(* CODESYS project MateusBastos_TalitaFelix (1).project

Project tree, tasks and I/O mapping:
  Device : CODESYS Control Win V3, 3S - Smart Software Solutions GmbH, order no. 305021, version 3.5.11.40
    application Application
      libraries: Standard, * (System)
      task MainTask (cyclic, interval t#10ms, priority 1) calls Main, Doca2_automatico, Doca1_manual, Doca2_manual, Doca1_automatico
      task Simulacao (cyclic, interval t#20ms, priority 1) calls Simulacao_Valores, Doca2_Simulacao, Gasolina_Simulacao, Doca1_Simulacao
      program Doca1_manual [SFC]
      global variables GVL
      program Doca2_manual [SFC]
      program Doca1_automatico [SFC]
      program Doca2_automatico [SFC]
      program Main [ST]
      Simulacao/
        program Doca2_Simulacao [ST]
        program Simulacao_Valores [ST]
        program Doca1_Simulacao [ST]
        program Gasolina_Simulacao [ST]
      program Emergencia [ST]
*)

// Device/Application/GVL
{attribute 'qualified_only'}
VAR_GLOBAL
// Sensores Analógicos - Entradas
LT_S01 : REAL;   // Sensor de porcentagem de etanol no silo 1
LT_S02 : REAL;   // Sensor de porcentagem de gasolina no silo 2
LT_S03 : REAL;   // Sensor de porcentagem de etanol no silo 3

// Sensores Discretos - Entradas
LSH_S01 : BOOL;  // Sensor de quantidade alta de combustível no silo 1
LSL_S01 : BOOL;  // Sensor de quantidade baixa de combustível no silo 1
LSH_S02 : BOOL;  // Sensor de quantidade alta de combustível no silo 2
LSL_S02 : BOOL;  // Sensor de quantidade baixa de combustível no silo 2
LSH_S03 : BOOL;  // Sensor de quantidade alta de combustível no silo 3
LSL_S03 : BOOL;  // Sensor de quantidade baixa de combustível no silo 3

// Atuadores Discretos - Saídas
VA_S01 : BOOL;   // Válvula de admissão de etanol no silo 1
VA_S02 : BOOL;   // Válvula de admissão de gasolina no silo 2
VA_S03 : BOOL;   // Válvula de admissão de etanol no silo 3
VS_S01 : BOOL;   // Válvula de admissão de etanol no tanque
VS_S02_1 : BOOL; // Válvula de admissão de gasolina no tanque (primeira seção)
VS_S02_2 : BOOL; // Válvula de admissão de gasolina no tanque (segunda seção)
VS_S03 : BOOL;   // Válvula de admissão de etanol no tanque
VC_TQ2 : BOOL;   // Válvula de saída do combustível para a mangueira (tanque 2)
VC_TQ1 : BOOL;   // Válvula de saída do combustível para a mangueira (tanque 1)
M1 : BOOL;       // Misturador 1
M2 : BOOL;       // Misturador 2
B_R1 : BOOL;     // Bomba de Etanol
B_R2 : BOOL;     // Bomba de Gasolina
C_D1 : BOOL;     // Cancela 1
C_D2 : BOOL;     // Cancela 2

// Interface - máquina
liga_manual: BOOL;
liga_auto: BOOL;
desliga: BOOL;
emergencia: BOOL;
rearme: BOOL;
Y_C_D1: BOOL;
Y_M_D1: BOOL;
Y_C_D2: BOOL;
Y_M_D2: BOOL;
etanol_D1: BOOL;
gasolina_p_D1: BOOL;
gasolina_n_D1: BOOL;
etanol_D2: BOOL;
gasolina_p_D2: BOOL;
gasolina_n_D2: BOOL;
//etanol_cheio: BOOL;
//gasolina_cheio: BOOL;
//timer_misturador: BOOL;
caminhao1_cheio: BOOL;
caminhao2_cheio: BOOL;
alarme_D1: BOOL;
alarme_D2: BOOL;

V_R_Etanol : INT := 200; //Vazao Reservatorio Etanol
V_R_Gasolina : INT := 200; //Vazao Reservatorio Gasolina
V_S01_TQ1 : INT := 100; // Vazão do Silo para o Tanque
V_S02_TQ : INT := 100; // Vazão DO Silo para o Tanque
V_S03_TQ2 : INT := 100; // Vazão DO Silo para o Tanque
TQ1_C : INT := 100;
TQ2_C : INT := 100;

volume_S01 : REAL := 50000;
volume_S02 : REAL := 50000;
volume_S03 : REAL := 50000;

volume_C1 : REAL := 0;
volume_C2 : REAL := 0;

volume_TQ1 : REAL := 0;
volume_TQ2 : REAL := 0;

volume_gasolina_C1 : REAL := 0;
volume_gasolina_C2 : REAL := 0;

volume_etanol_C1 : REAL := 0;
volume_etanol_C2 : REAL := 0;

PREMIUM : BOOL; // SE PREMIUM, GASOLINA PREMIUM.
ETANOL : BOOL; //EXCLUIR ESSA VARIAVEL

modo_op : BOOL; //Modo de operação atual do programa
switch : BOOl; //Modo de operação que o operador definiu

END_VAR

// Device/Application/Main
PROGRAM Main


// Desliga foi ativado
IF GVL.desliga THEN
	// Para a operação de todas as docas
	Doca1_manual.Ligar := FALSE;
	Doca2_manual.Ligar := FALSE;
	Doca1_automatico.Ligar := FALSE;
	Doca2_automatico.Ligar := FALSE;

// Emergência foi ativada
ELSIF GVL.emergencia AND NOT GVL.Rearme AND NOT GVL.modo_op THEN
	// Para a operação de todas as docas
	Emergencia.Ligar := TRUE;
	Doca1_manual.Ligar := FALSE;
	Doca2_manual.Ligar := FALSE;

ELSIF GVL.rearme AND NOT GVL.modo_op THEN
	Emergencia.Ligar := FALSE;
	Doca1_manual.Ligar := TRUE;
	Doca2_manual.Ligar := TRUE;

ELSIF GVL.emergencia AND NOT GVL.Rearme AND GVL.modo_op THEN
	// Para a operação de todas as docas
	Emergencia.Ligar := TRUE;
	Doca1_automatico.Ligar := FALSE;
	Doca2_automatico.Ligar := FALSE;

ELSIF GVL.rearme AND GVL.modo_op THEN
	Emergencia.Ligar := FALSE;
	Doca1_automatico.Ligar := TRUE;
	Doca2_automatico.Ligar := TRUE;

// Seleção do modo de operação e liga	
ELSE
	// Se o modo de operação for manual e o operador requisitar o modo automático, o modo_op será trocado se não houver caminhões na doca e todas as válvulas estiverem fechadas
	IF GVL.modo_op = 0 AND GVL.switch = 1 THEN
		IF (Doca1_manual.Init.x AND Doca2_manual.Init.x) OR (NOT Doca1_manual.Ligar AND NOT Doca2_manual.Ligar) OR Emergencia.Ligar THEN
			GVL.modo_op := 1;
		END_IF	
	END_IF
	
	// Se o modo de operação for automático e o operador requisitar o modo manual, o modo_op será trocado se o processo estiver desligago ou em estado de emergência
	IF GVL.modo_op = 1 AND GVL.switch = 0 THEN
		IF NOT GVL.liga_auto OR Emergencia.Ligar THEN
			GVL.modo_op := 0;
		END_IF	
	END_IF
	
	IF GVL.liga_manual AND NOT GVL.modo_op THEN
		// Inicia a operação manual das duas docas
		Doca1_manual.Ligar := TRUE;
		Doca2_manual.Ligar := TRUE;
		Doca1_automatico.Ligar := FALSE;
		Doca2_automatico.Ligar := FALSE;
		
	ELSIF GVL.liga_auto AND GVL.modo_op THEN
		// Inicia a operação automática das duas docas
		Doca1_manual.Ligar := FALSE;
		Doca2_manual.Ligar := FALSE;
		Doca1_automatico.Ligar := TRUE;
		Doca2_automatico.Ligar := TRUE;
		
	END_IF
END_IF

END_PROGRAM

// Device/Application/Doca1_manual
PROGRAM Doca1_manual
VAR_INPUT
	Ligar : BOOL;
END_VAR

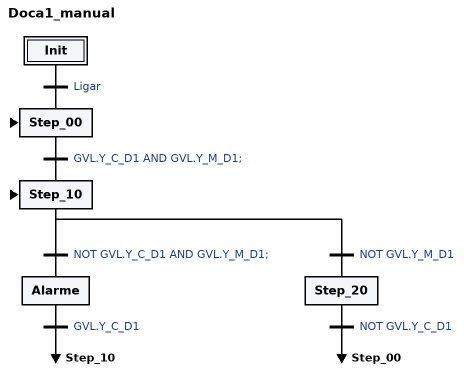
INITIAL_STEP Init:
END_STEP
TRANSITION FROM Init TO Step_00
    := Ligar;
END_TRANSITION
STEP Step_00:
END_STEP
TRANSITION FROM Step_00 TO Step_10
    := GVL.Y_C_D1 AND GVL.Y_M_D1;
END_TRANSITION
STEP Step_10:
END_STEP
TRANSITION FROM Step_10 TO Alarme
    := NOT GVL.Y_C_D1 AND GVL.Y_M_D1;
END_TRANSITION
STEP Alarme:
END_STEP
TRANSITION FROM Alarme TO Step_10
    := GVL.Y_C_D1;
END_TRANSITION
TRANSITION FROM Step_10 TO Step_20
    := NOT GVL.Y_M_D1;
END_TRANSITION
STEP Step_20:
END_STEP
TRANSITION FROM Step_20 TO Step_00
    := NOT GVL.Y_C_D1;
END_TRANSITION

END_PROGRAM

// Device/Application/Doca2_manual
PROGRAM Doca2_manual
VAR_INPUT
	Ligar : BOOL;
END_VAR

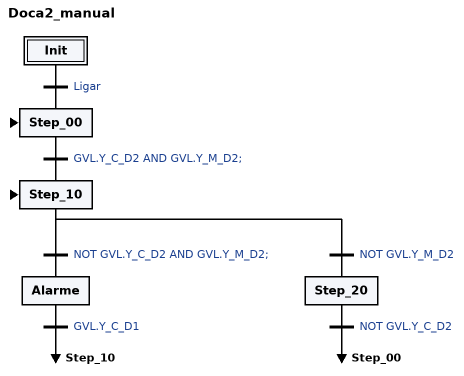
INITIAL_STEP Init:
END_STEP
TRANSITION FROM Init TO Step_00
    := Ligar;
END_TRANSITION
STEP Step_00:
END_STEP
TRANSITION FROM Step_00 TO Step_10
    := GVL.Y_C_D2 AND GVL.Y_M_D2;
END_TRANSITION
STEP Step_10:
END_STEP
TRANSITION FROM Step_10 TO Alarme
    := NOT GVL.Y_C_D2 AND GVL.Y_M_D2;
END_TRANSITION
STEP Alarme:
END_STEP
TRANSITION FROM Alarme TO Step_10
    := GVL.Y_C_D1;
END_TRANSITION
TRANSITION FROM Step_10 TO Step_20
    := NOT GVL.Y_M_D2;
END_TRANSITION
STEP Step_20:
END_STEP
TRANSITION FROM Step_20 TO Step_00
    := NOT GVL.Y_C_D2;
END_TRANSITION

END_PROGRAM

// Device/Application/Doca1_automatico
	PROGRAM Doca1_automatico

VAR_INPUT
	Ligar : BOOL;
	etanol_cheio: BOOL;
	gasolina_cheio: BOOL;
END_VAR

VAR
	
END_VAR

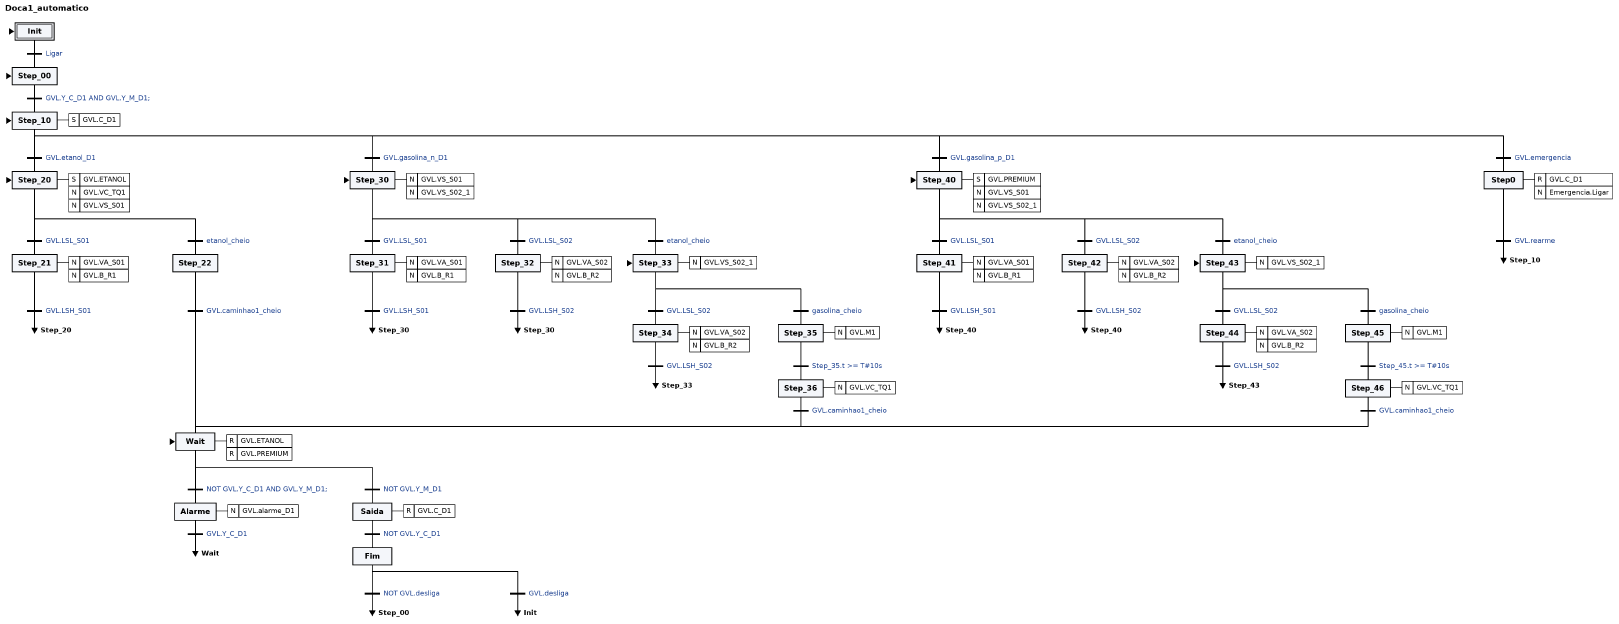
INITIAL_STEP Init:
END_STEP
TRANSITION FROM Init TO Step_00
    := Ligar;
END_TRANSITION
STEP Step_00:
END_STEP
TRANSITION FROM Step_00 TO Step_10
    := GVL.Y_C_D1 AND GVL.Y_M_D1;
END_TRANSITION
STEP Step_10:
    GVL.C_D1(S);
END_STEP
TRANSITION FROM Step_10 TO Step_20
    := GVL.etanol_D1;
END_TRANSITION
STEP Step_20:
    GVL.ETANOL(S);
    GVL.VC_TQ1(N);
    GVL.VS_S01(N);
END_STEP
TRANSITION FROM Step_20 TO Step_21
    := GVL.LSL_S01;
END_TRANSITION
STEP Step_21:
    GVL.VA_S01(N);
    GVL.B_R1(N);
END_STEP
TRANSITION FROM Step_21 TO Step_20
    := GVL.LSH_S01;
END_TRANSITION
TRANSITION FROM Step_20 TO Step_22
    := etanol_cheio;
END_TRANSITION
STEP Step_22:
END_STEP
TRANSITION FROM Step_22 TO Wait
    := GVL.caminhao1_cheio;
END_TRANSITION
TRANSITION FROM Step_10 TO Step_30
    := GVL.gasolina_n_D1;
END_TRANSITION
STEP Step_30:
    GVL.VS_S01(N);
    GVL.VS_S02_1(N);
END_STEP
TRANSITION FROM Step_30 TO Step_31
    := GVL.LSL_S01;
END_TRANSITION
STEP Step_31:
    GVL.VA_S01(N);
    GVL.B_R1(N);
END_STEP
TRANSITION FROM Step_31 TO Step_30
    := GVL.LSH_S01;
END_TRANSITION
TRANSITION FROM Step_30 TO Step_32
    := GVL.LSL_S02;
END_TRANSITION
STEP Step_32:
    GVL.VA_S02(N);
    GVL.B_R2(N);
END_STEP
TRANSITION FROM Step_32 TO Step_30
    := GVL.LSH_S02;
END_TRANSITION
TRANSITION FROM Step_30 TO Step_33
    := etanol_cheio;
END_TRANSITION
STEP Step_33:
    GVL.VS_S02_1(N);
END_STEP
TRANSITION FROM Step_33 TO Step_34
    := GVL.LSL_S02;
END_TRANSITION
STEP Step_34:
    GVL.VA_S02(N);
    GVL.B_R2(N);
END_STEP
TRANSITION FROM Step_34 TO Step_33
    := GVL.LSH_S02;
END_TRANSITION
TRANSITION FROM Step_33 TO Step_35
    := gasolina_cheio;
END_TRANSITION
STEP Step_35:
    GVL.M1(N);
END_STEP
TRANSITION FROM Step_35 TO Step_36
    := Step_35.t >= T#10s;
END_TRANSITION
STEP Step_36:
    GVL.VC_TQ1(N);
END_STEP
TRANSITION FROM Step_36 TO Wait
    := GVL.caminhao1_cheio;
END_TRANSITION
TRANSITION FROM Step_10 TO Step_40
    := GVL.gasolina_p_D1;
END_TRANSITION
STEP Step_40:
    GVL.PREMIUM(S);
    GVL.VS_S01(N);
    GVL.VS_S02_1(N);
END_STEP
TRANSITION FROM Step_40 TO Step_41
    := GVL.LSL_S01;
END_TRANSITION
STEP Step_41:
    GVL.VA_S01(N);
    GVL.B_R1(N);
END_STEP
TRANSITION FROM Step_41 TO Step_40
    := GVL.LSH_S01;
END_TRANSITION
TRANSITION FROM Step_40 TO Step_42
    := GVL.LSL_S02;
END_TRANSITION
STEP Step_42:
    GVL.VA_S02(N);
    GVL.B_R2(N);
END_STEP
TRANSITION FROM Step_42 TO Step_40
    := GVL.LSH_S02;
END_TRANSITION
TRANSITION FROM Step_40 TO Step_43
    := etanol_cheio;
END_TRANSITION
STEP Step_43:
    GVL.VS_S02_1(N);
END_STEP
TRANSITION FROM Step_43 TO Step_44
    := GVL.LSL_S02;
END_TRANSITION
STEP Step_44:
    GVL.VA_S02(N);
    GVL.B_R2(N);
END_STEP
TRANSITION FROM Step_44 TO Step_43
    := GVL.LSH_S02;
END_TRANSITION
TRANSITION FROM Step_43 TO Step_45
    := gasolina_cheio;
END_TRANSITION
STEP Step_45:
    GVL.M1(N);
END_STEP
TRANSITION FROM Step_45 TO Step_46
    := Step_45.t >= T#10s;
END_TRANSITION
STEP Step_46:
    GVL.VC_TQ1(N);
END_STEP
TRANSITION FROM Step_46 TO Wait
    := GVL.caminhao1_cheio;
END_TRANSITION
TRANSITION FROM Step_10 TO Step0
    := GVL.emergencia;
END_TRANSITION
STEP Step0:
    GVL.C_D1(R);
    Emergencia.Ligar(N);
END_STEP
TRANSITION FROM Step0 TO Step_10
    := GVL.rearme;
END_TRANSITION
STEP Wait:
    GVL.ETANOL(R);
    GVL.PREMIUM(R);
END_STEP
TRANSITION FROM Wait TO Alarme
    := NOT GVL.Y_C_D1 AND GVL.Y_M_D1;
END_TRANSITION
STEP Alarme:
    GVL.alarme_D1(N);
END_STEP
TRANSITION FROM Alarme TO Wait
    := GVL.Y_C_D1;
END_TRANSITION
TRANSITION FROM Wait TO Saida
    := NOT GVL.Y_M_D1;
END_TRANSITION
STEP Saida:
    GVL.C_D1(R);
END_STEP
TRANSITION FROM Saida TO Fim
    := NOT GVL.Y_C_D1;
END_TRANSITION
STEP Fim:
END_STEP
TRANSITION FROM Fim TO Step_00
    := NOT GVL.desliga;
END_TRANSITION
TRANSITION FROM Fim TO Init
    := GVL.desliga;
END_TRANSITION

END_PROGRAM

// Device/Application/Doca2_automatico
PROGRAM Doca2_automatico
VAR_INPUT
	Ligar : BOOL;
	etanol_cheio: BOOL;
	gasolina_cheio: BOOL;
END_VAR

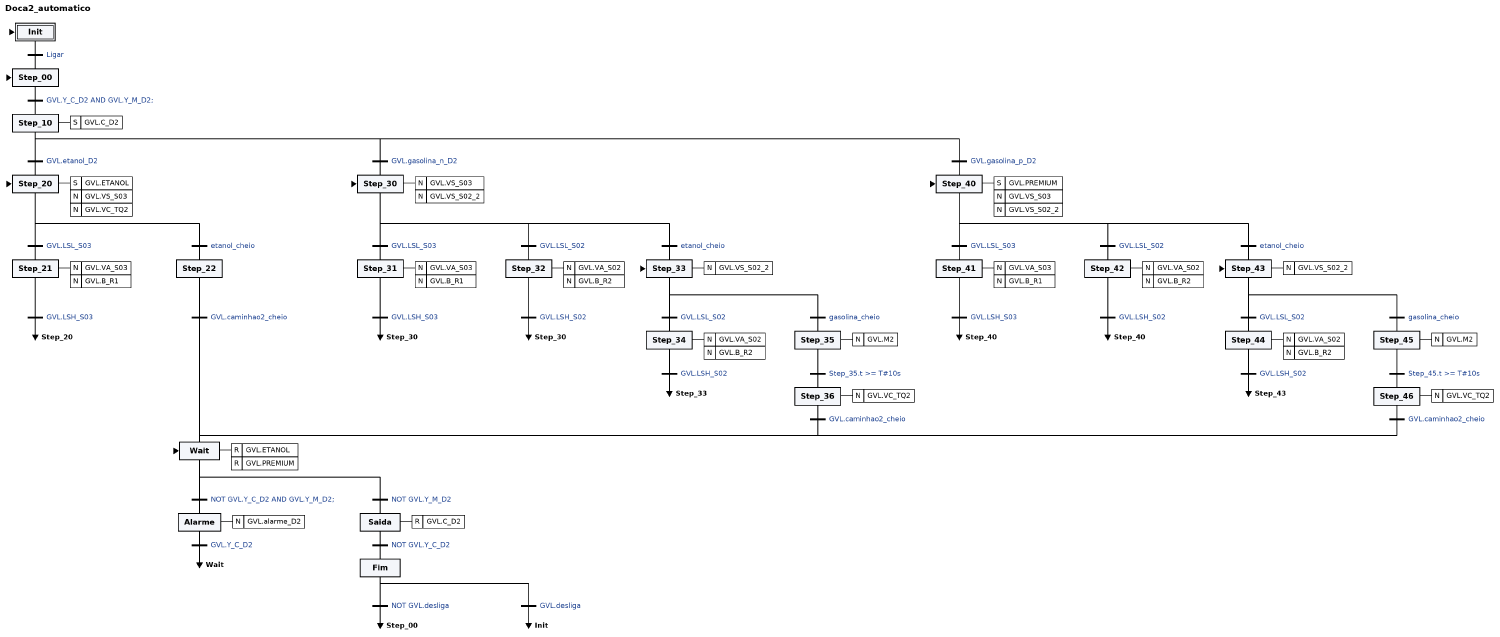
INITIAL_STEP Init:
END_STEP
TRANSITION FROM Init TO Step_00
    := Ligar;
END_TRANSITION
STEP Step_00:
END_STEP
TRANSITION FROM Step_00 TO Step_10
    := GVL.Y_C_D2 AND GVL.Y_M_D2;
END_TRANSITION
STEP Step_10:
    GVL.C_D2(S);
END_STEP
TRANSITION FROM Step_10 TO Step_20
    := GVL.etanol_D2;
END_TRANSITION
STEP Step_20:
    GVL.ETANOL(S);
    GVL.VS_S03(N);
    GVL.VC_TQ2(N);
END_STEP
TRANSITION FROM Step_20 TO Step_21
    := GVL.LSL_S03;
END_TRANSITION
STEP Step_21:
    GVL.VA_S03(N);
    GVL.B_R1(N);
END_STEP
TRANSITION FROM Step_21 TO Step_20
    := GVL.LSH_S03;
END_TRANSITION
TRANSITION FROM Step_20 TO Step_22
    := etanol_cheio;
END_TRANSITION
STEP Step_22:
END_STEP
TRANSITION FROM Step_22 TO Wait
    := GVL.caminhao2_cheio;
END_TRANSITION
TRANSITION FROM Step_10 TO Step_30
    := GVL.gasolina_n_D2;
END_TRANSITION
STEP Step_30:
    GVL.VS_S03(N);
    GVL.VS_S02_2(N);
END_STEP
TRANSITION FROM Step_30 TO Step_31
    := GVL.LSL_S03;
END_TRANSITION
STEP Step_31:
    GVL.VA_S03(N);
    GVL.B_R1(N);
END_STEP
TRANSITION FROM Step_31 TO Step_30
    := GVL.LSH_S03;
END_TRANSITION
TRANSITION FROM Step_30 TO Step_32
    := GVL.LSL_S02;
END_TRANSITION
STEP Step_32:
    GVL.VA_S02(N);
    GVL.B_R2(N);
END_STEP
TRANSITION FROM Step_32 TO Step_30
    := GVL.LSH_S02;
END_TRANSITION
TRANSITION FROM Step_30 TO Step_33
    := etanol_cheio;
END_TRANSITION
STEP Step_33:
    GVL.VS_S02_2(N);
END_STEP
TRANSITION FROM Step_33 TO Step_34
    := GVL.LSL_S02;
END_TRANSITION
STEP Step_34:
    GVL.VA_S02(N);
    GVL.B_R2(N);
END_STEP
TRANSITION FROM Step_34 TO Step_33
    := GVL.LSH_S02;
END_TRANSITION
TRANSITION FROM Step_33 TO Step_35
    := gasolina_cheio;
END_TRANSITION
STEP Step_35:
    GVL.M2(N);
END_STEP
TRANSITION FROM Step_35 TO Step_36
    := Step_35.t >= T#10s;
END_TRANSITION
STEP Step_36:
    GVL.VC_TQ2(N);
END_STEP
TRANSITION FROM Step_36 TO Wait
    := GVL.caminhao2_cheio;
END_TRANSITION
TRANSITION FROM Step_10 TO Step_40
    := GVL.gasolina_p_D2;
END_TRANSITION
STEP Step_40:
    GVL.PREMIUM(S);
    GVL.VS_S03(N);
    GVL.VS_S02_2(N);
END_STEP
TRANSITION FROM Step_40 TO Step_41
    := GVL.LSL_S03;
END_TRANSITION
STEP Step_41:
    GVL.VA_S03(N);
    GVL.B_R1(N);
END_STEP
TRANSITION FROM Step_41 TO Step_40
    := GVL.LSH_S03;
END_TRANSITION
TRANSITION FROM Step_40 TO Step_42
    := GVL.LSL_S02;
END_TRANSITION
STEP Step_42:
    GVL.VA_S02(N);
    GVL.B_R2(N);
END_STEP
TRANSITION FROM Step_42 TO Step_40
    := GVL.LSH_S02;
END_TRANSITION
TRANSITION FROM Step_40 TO Step_43
    := etanol_cheio;
END_TRANSITION
STEP Step_43:
    GVL.VS_S02_2(N);
END_STEP
TRANSITION FROM Step_43 TO Step_44
    := GVL.LSL_S02;
END_TRANSITION
STEP Step_44:
    GVL.VA_S02(N);
    GVL.B_R2(N);
END_STEP
TRANSITION FROM Step_44 TO Step_43
    := GVL.LSH_S02;
END_TRANSITION
TRANSITION FROM Step_43 TO Step_45
    := gasolina_cheio;
END_TRANSITION
STEP Step_45:
    GVL.M2(N);
END_STEP
TRANSITION FROM Step_45 TO Step_46
    := Step_45.t >= T#10s;
END_TRANSITION
STEP Step_46:
    GVL.VC_TQ2(N);
END_STEP
TRANSITION FROM Step_46 TO Wait
    := GVL.caminhao2_cheio;
END_TRANSITION
STEP Wait:
    GVL.ETANOL(R);
    GVL.PREMIUM(R);
END_STEP
TRANSITION FROM Wait TO Alarme
    := NOT GVL.Y_C_D2 AND GVL.Y_M_D2;
END_TRANSITION
STEP Alarme:
    GVL.alarme_D2(N);
END_STEP
TRANSITION FROM Alarme TO Wait
    := GVL.Y_C_D2;
END_TRANSITION
TRANSITION FROM Wait TO Saida
    := NOT GVL.Y_M_D2;
END_TRANSITION
STEP Saida:
    GVL.C_D2(R);
END_STEP
TRANSITION FROM Saida TO Fim
    := NOT GVL.Y_C_D2;
END_TRANSITION
STEP Fim:
END_STEP
TRANSITION FROM Fim TO Step_00
    := NOT GVL.desliga;
END_TRANSITION
TRANSITION FROM Fim TO Init
    := GVL.desliga;
END_TRANSITION

END_PROGRAM

// Device/Application/Emergencia
PROGRAM Emergencia

VAR_INPUT
	Ligar : BOOL;
END_VAR

IF Ligar THEN
	GVL.VA_S01 := FALSE;   
	GVL.VA_S02 := FALSE;
	GVL.VA_S03 := FALSE;
	GVL.VS_S01 := FALSE;
	GVL.VS_S02_1 := FALSE;
	GVL.VS_S02_2 := FALSE;
	GVL.VS_S03 := FALSE;
	GVL.VC_TQ2 := FALSE;
	GVL.VC_TQ1 := FALSE;
	GVL.M1 := FALSE;
	GVL.M2 := FALSE;
	GVL.B_R1 := FALSE;
	//GVL.B_R2 := FALSE;
END_IF

END_PROGRAM

// Device/Application/Simulacao/Simulacao_Valores
PROGRAM Simulacao_Valores
VAR
	Volume_gasolina_comum : REAL := 25000 * 0.75;
	Volume_etanol_comum : REAL := 25000 * 0.25;
	Volume_gasolina_premium : REAL := 25000 * 0.73;
	Volume_etanol_premium : REAL := 25000 * 0.27;
END_VAR

IF GVL.volume_C1 >= 25000 THEN//AND GVL.volume_gasolina_C1 = 0 THEN
	Doca1_automatico.etanol_cheio := TRUE;
	GVL.caminhao1_cheio := TRUE;
	
	GVL.volume_etanol_C1 := 0;
	GVL.volume_gasolina_C1 := 0;
	
ELSIF GVL.volume_S01 <= 5000 THEN
	GVL.LSL_S01 := TRUE;
	GVL.LSH_S01 := FALSE;
	
ELSIF  GVL.volume_S02 <= 5000 THEN
	GVL.LSL_S02 := TRUE;
	GVL.LSH_S02 := FALSE;

ELSIF GVL.volume_S02 >= 45000 THEN
	GVL.LSH_S02 := TRUE;
	GVL.LSL_S02 := FALSE;
	
ELSIF GVL.volume_S01 >= 45000 THEN
	GVL.LSH_S01 := TRUE;
	GVL.LSL_S01 := FALSE;

ELSIF GVL.volume_etanol_C1 >= Volume_etanol_premium AND NOT (GVL.volume_gasolina_C1 >= Volume_gasolina_premium) AND GVL.PREMIUM THEN // PODE GERAR UM FUTURO PROBLEMA
	Doca1_automatico.etanol_cheio := TRUE;
	
ELSIF GVL.volume_gasolina_C1 >= Volume_gasolina_premium AND NOT GVL.M1 AND GVL.PREMIUM THEN // PODE GERAR UM PROBLEMA NO FUTURO
	Doca1_automatico.gasolina_cheio := TRUE;	
	
ELSIF GVL.volume_etanol_C1 >= Volume_etanol_comum AND NOT (GVL.volume_gasolina_C1 >= Volume_gasolina_comum) AND NOT GVL.PREMIUM THEN // PODE GERAR UM FUTURO PROBLEMA
	Doca1_automatico.etanol_cheio := TRUE;
	
ELSIF GVL.volume_gasolina_C1 >= Volume_gasolina_comum AND NOT GVL.M1 AND NOT GVL.PREMIUM THEN // PODE GERAR UM PROBLEMA NO FUTURO
	Doca1_automatico.gasolina_cheio := TRUE;
	
ELSIF GVL.M1 THEN
	GVL.volume_etanol_C1 := 0;
	GVL.volume_gasolina_C1 := 0;
	
ELSE
	GVL.LSL_S01 := FALSE;
	GVL.caminhao1_cheio := FALSE;
	Doca1_automatico.gasolina_cheio := FALSE;
	Doca1_automatico.etanol_cheio := FALSE;
	GVL.LSH_S01 := FALSE;
END_IF

END_PROGRAM

// Device/Application/Simulacao/Doca2_Simulacao
PROGRAM Doca2_Simulacao
VAR
END_VAR

IF NOT GVL.emergencia THEN
	//Estado  20 & //Estado 31 & //Estado 41 & //Estado 34 & //Estado 44
	IF GVL.VA_S03 AND GVL.B_R1 AND GVL.C_D2 THEN
	// Enchendo o Silo 01 de Etanol - STEP_21
		GVL.volume_S03 := GVL.volume_S03 + GVL.V_R_Etanol;
	
		GVL.volume_TQ2 := GVL.volume_TQ2;
		
		GVL.volume_C2 := GVL.volume_C2;
		
	//Estado  20	
	ELSIF GVL.VA_S02 AND GVL.B_R2 AND (GVL.ETANOL OR NOT GVL.Y_C_D1) THEN // Caso em que o somente a doca 2 está utilizando gasolina
		GVL.volume_S02 := GVL.volume_S02 + GVL.V_R_Gasolina;
		
	ELSIF GVL.VS_S03 AND GVL.C_D2 AND NOT GVL.VS_S02_2 AND GVL.VC_TQ2 THEN
	// Enchendo o Tanque 1 & Esvaziando o Silo 01 - STEP_20
		GVL.volume_S03 := GVL.volume_S03 - GVL.V_S03_TQ2;
		
		GVL.volume_TQ2 := GVL.volume_TQ2 + GVL.TQ2_C - GVL.V_S03_TQ2;
		
		GVL.volume_C2 := GVL.volume_C2 + GVL.TQ2_C;
		
	//Estado 30	- STEP_30 e STEP_40
	ELSIF GVL.VS_S03 AND GVL.VS_S02_2 AND GVL.C_D2 THEN
	// Enchendo o TQ 1 && Esvaziando o Silo 01 && Esvaziando o Silo 02
	
	//Situação em que começo a encher o tanque de gasolina e de etanol simultaneamente
	
		GVL.volume_S03 := GVL.volume_S03 - GVL.V_S03_TQ2; // Diminuo o volume do Silo 3
		
		GVL.volume_S02 := GVL.volume_S02 - GVL.V_S02_TQ; // Diminuo o volume do Silo 2
		
		GVL.volume_C2 := GVL.volume_C2; // Mantenho o volume do caminhão constante
		
		GVL.volume_TQ2 := GVL.volume_TQ2 + GVL.V_S02_TQ + GVL.V_S03_TQ2; // Aumento o volume do tanque 1
		
		GVL.volume_gasolina_C2 := GVL.volume_gasolina_C2 + GVL.V_S02_TQ; // Aumento a contagem da gasolina que está entrando no tanque
		
		GVL.volume_etanol_C2 := GVL.volume_etanol_C2 + GVL.V_S03_TQ2; // Aumento a contagem de etanol que está entrando no tanque
		
	//Estado 33 & Estado 43 - STEP_33
	ELSIF GVL.VS_S02_2 AND NOT GVL.VC_TQ2 AND GVL.C_D2 THEN
		GVL.volume_S02 := GVL.volume_S02 - GVL.V_S02_TQ;	
		
		GVL.volume_C2 := GVL.volume_C2;
		
		GVL.volume_TQ2 := GVL.volume_TQ2 + GVL.V_S02_TQ;
		
		GVL.volume_gasolina_C2 := GVL.volume_gasolina_C2 + GVL.V_S02_TQ;
		
	//Estado 35 & //Estado 45
	ELSIF GVL.M2 AND GVL.C_D2 THEN
		GVL.volume_C2 := GVL.volume_C2;
		GVL.volume_TQ2 := GVL.volume_TQ2;
		
	//Estado 36 & //Estado 46
	ELSIF GVL.VC_TQ2 AND GVL.C_D2 THEN
		GVL.volume_C2 := GVL.volume_C2 + GVL.TQ2_C;
		GVL.volume_TQ2 := GVL.volume_TQ2 - GVL.TQ2_C;
	
	ELSIF NOT GVL.Y_C_D2 AND GVL.C_D2 THEN 
		GVL.volume_C2 := 0;
		GVL.volume_TQ2 := 0;
	
	END_IF
END_IF

END_PROGRAM

// Device/Application/Simulacao/Gasolina_Simulacao
PROGRAM Gasolina_Simulacao
VAR
	Volume_gasolina_comum : REAL := 25000 * 0.75;
	Volume_etanol_comum : REAL := 25000 * 0.25;
	Volume_gasolina_premium : REAL := 25000 * 0.73;
	Volume_etanol_premium : REAL := 25000 * 0.27;
END_VAR

IF GVL.volume_C2 >= 25000 THEN // AND GVL.volume_gasolina_C2 = 0 THEN
	Doca2_automatico.etanol_cheio := TRUE;
	GVL.caminhao2_cheio := TRUE;
	
	GVL.volume_etanol_C2 := 0;
	GVL.volume_gasolina_C2 := 0;
	
ELSIF GVL.volume_S03 <= 5000 THEN
	GVL.LSL_S03 := TRUE;
	GVL.LSH_S03 := FALSE;

ELSIF  GVL.volume_S02 <= 5000 THEN
	GVL.LSL_S02 := TRUE;
	GVL.LSH_S02 := FALSE;

ELSIF GVL.volume_S02 >= 45000 THEN
	GVL.LSH_S02 := TRUE;
	GVL.LSL_S02 := FALSE;
	
ELSIF GVL.volume_S03 >= 45000 THEN
	GVL.LSH_S03 := TRUE;
	GVL.LSL_S03 := FALSE;

ELSIF GVL.volume_etanol_C2 >= Volume_etanol_premium AND NOT (GVL.volume_gasolina_C2 >= Volume_gasolina_premium) AND GVL.PREMIUM THEN // PODE GERAR UM FUTURO PROBLEMA
	Doca2_automatico.etanol_cheio := TRUE;	
	
ELSIF GVL.volume_gasolina_C2 >= Volume_gasolina_premium AND NOT GVL.M2 AND GVL.PREMIUM THEN // PODE GERAR UM PROBLEMA NO FUTURO	
	Doca2_automatico.gasolina_cheio := TRUE;
	
ELSIF GVL.volume_etanol_C2 >= Volume_etanol_comum AND NOT (GVL.volume_gasolina_C2 >= Volume_gasolina_comum) AND NOT GVL.PREMIUM THEN // PODE GERAR UM FUTURO PROBLEMA
	Doca2_automatico.etanol_cheio := TRUE;
	
ELSIF GVL.volume_gasolina_C2 >= Volume_gasolina_comum AND NOT GVL.M2 AND NOT GVL.PREMIUM THEN // PODE GERAR UM PROBLEMA NO FUTURO
	Doca2_automatico.gasolina_cheio := TRUE;
	
ELSIF GVL.M2 THEN
	GVL.volume_etanol_C2 := 0;
	GVL.volume_gasolina_C2 := 0;
	
ELSE
	GVL.LSL_S03 := FALSE;
	GVL.caminhao2_cheio := FALSE;
	Doca2_automatico.etanol_cheio := FALSE;
	Doca2_automatico.gasolina_cheio := FALSE;
	GVL.LSH_S03 := FALSE;
END_IF

END_PROGRAM

// Device/Application/Simulacao/Doca1_Simulacao
PROGRAM Doca1_Simulacao
VAR
END_VAR

IF NOT GVL.emergencia THEN
	//Estado  20 & //Estado 31 & //Estado 41 & //Estado 34 & //Estado 44
	IF GVL.VA_S01 AND GVL.B_R1 AND GVL.C_D1 THEN
	// Enchendo o Silo 01 de Etanol - STEP_21
		GVL.volume_S01 := GVL.volume_S01 + GVL.V_R_Etanol;
	
		GVL.volume_TQ1 := GVL.volume_TQ1;
		
		GVL.volume_C1 := GVL.volume_C1;
		
	ELSIF GVL.VA_S02 AND GVL.B_R2 THEN
	// Enchendo o Silo de Gasolina
		GVL.volume_S02 := GVL.volume_S02 + GVL.V_R_Gasolina;
	
	//Estado  21	
	ELSIF GVL.VS_S01 AND GVL.C_D1 AND NOT GVL.VS_S02_1 AND GVL.VC_TQ1 THEN
	// Enchendo o Tanque 1 & Esvaziando o Silo 01 - STEP_20
		GVL.volume_S01 := GVL.volume_S01 - GVL.V_S01_TQ1;
		
		GVL.volume_TQ1 := GVL.volume_TQ1 + GVL.TQ1_C - GVL.V_S01_TQ1;
		
		GVL.volume_C1 := GVL.volume_C1 + GVL.TQ1_C;
		
	//Estado 30	- STEP_30
	ELSIF GVL.VS_S01 AND GVL.VS_S02_1 AND GVL.C_D1 THEN
	// Enchendo o TQ 1 && Esvaziando o Silo 01 && Esvaziando o Silo 02
	
	//Situação em que começo a encher o tanque de gasolina e de etanol simultaneamente
	
		GVL.volume_S01 := GVL.volume_S01 - GVL.V_S01_TQ1; // Diminuo o volume do Silo 1
		
		GVL.volume_S02 := GVL.volume_S02 - GVL.V_S02_TQ; // Diminuo o volume do Silo 2
		
		GVL.volume_C1 := GVL.volume_C1; // Mantenho o volume do caminhão constante
		
		GVL.volume_TQ1 := GVL.volume_TQ1 + GVL.V_S02_TQ + GVL.V_S01_TQ1; // Aumento o volume do tanque 1
		
		GVL.volume_gasolina_C1 := GVL.volume_gasolina_C1 + GVL.V_S02_TQ; // Aumento a contagem da gasolina que está entrando no tanque
		
		GVL.volume_etanol_C1 := GVL.volume_etanol_C1 + GVL.V_S01_TQ1; // Aumento a contagem de etanol que está entrando no tanque
		
	//Estado 33 & Estado 43 - STEP_33
	ELSIF GVL.VS_S02_1 AND NOT GVL.VC_TQ1 AND GVL.C_D1 THEN
		GVL.volume_S02 := GVL.volume_S02 - GVL.V_S02_TQ;	
		
		GVL.volume_C1 := GVL.volume_C1;
		
		GVL.volume_TQ1 := GVL.volume_TQ1 + GVL.V_S02_TQ;
		
		GVL.volume_gasolina_C1 := GVL.volume_gasolina_C1 + GVL.V_S02_TQ;
		
	//Estado 35 & //Estado 45
	ELSIF GVL.M1 AND GVL.C_D1 THEN
		GVL.volume_C1 := GVL.volume_C1;
		GVL.volume_TQ1 := GVL.volume_TQ1;
		
	//Estado 36 & //Estado 46
	ELSIF GVL.VC_TQ1 AND GVL.C_D1 THEN
		GVL.volume_C1 := GVL.volume_C1 + GVL.TQ1_C;
		GVL.volume_TQ1 := GVL.volume_TQ1 - GVL.TQ1_C;
	
	ELSIF NOT GVL.Y_C_D1 AND GVL.C_D1 THEN 
		GVL.volume_C1 := 0;
		GVL.volume_TQ1 := 0;
	END_IF
END_IF

END_PROGRAM
